# EPICS substitutions: edtPdvApp/camera_config/avtGoldEye008.substitutions
# A simple MODEL substitutions file which preserves macro defaults
# but expands any inluded rbvMonitor.template or other templates.
file avtGoldEye008.template
{
	{
		P				= "\$(P)",
		R				= "\$(R)",
		PORT			= "\$(PORT)",
		PWIDTH			= "\$(PWIDTH=TRIG:PULSE:WIDTH)",
		PW_SCALE		= "\$(PW_SCALE=1e9)",
		SerialDisable	= "\$(SerialDisable)"
	}
}
